// TIA Portal project "实验3_V20" (V20)

(* hardware
DEVICE "S7-300/ET200M station_1"  S7-300 station
   slot 0: "导轨_0"  Rail  6ES7 390-1***0-0AA0
   slot 2: "PLC_1"  CPU 314C-2 DP  6ES7 314-6CH04-0AB0  V3.3
      slot 0: "MPI 接口_1"  MPI
      slot 1: "DP 接口_1"  DP
      slot 2: "DI 24/DO 16_1"  DI24/DO16
      slot 3: "AI 5/AO 2_1"  AI5/AO2
      slot 4: "计数_1"  Counter
      slot 5: "定位_1"  Positioning
*)

// ===== PLC "PLC_1"  CPU 314C-2 DP =====

VAR_GLOBAL   // PLC tag table "默认变量表"
   "启动开关" AT %I0.0 : Bool;
   "光电传感器1" AT %I0.1 : Bool;
   "光电传感器2" AT %I0.2 : Bool;
   "光电传感器3" AT %I0.3 : Bool;
   "光电传感器4" AT %I0.4 : Bool;
   "电机正转" AT %Q4.1 : Bool;
   "电机反转" AT %Q4.2 : Bool;
   "位置1" AT %Q4.3 : Bool;
   "位置2" AT %Q4.4 : Bool;
   "位置3" AT %Q4.5 : Bool;
END_VAR

DATA_BLOCK "流程_DB"   // DB1
{ S7_Optimized_Access := 'FALSE' }
VERSION : 0.1
// stored: InstanceOfName 流程
"流程"
BEGIN
END_DATA_BLOCK

FUNCTION_BLOCK "流程"   // FB1, GRAPH
{ S7_Optimized_Access := 'FALSE' }
VERSION : 0.1
   VAR_INPUT
      OFF_SQ : Bool := false;   // 关闭顺控器
      INIT_SQ : Bool := false;   // 将顺序设置为初始状态
      ACK_EF : Bool := false;   // 确认所有的错误和故障
      S_PREV : Bool := false;   // 在S_NO输出参数中显示前导步
      S_NEXT : Bool := false;   // 在S_NO输出参数中显示后续步。
      SW_AUTO : Bool := false;   // 自动模式
      SW_TAP : Bool := false;   // 半自动/转换条件切换
      SW_TOP : Bool := false;   // 半自动/忽略转换条件
      SW_MAN : Bool := false;   // 手动模式
      S_SEL : Int := 0;   // 选择要在 S_NO中输出的步。
      S_ON : Bool := false;   // 激活S_NO 中显示的步。
      S_OFF : Bool := false;   // 禁用 S_NO 中标识的步
      T_PUSH : Bool := false;   // 允许在半自动模式下跳过转换条件。
   END_VAR
   VAR_OUTPUT
      S_NO : Int := 0;   // 步编号
      S_MORE : Bool := false;   // 更多步可用，并可在S_NO中显示。
      S_ACTIVE : Bool := false;   // 在S_NO 中显示的步是激活的。
      ERR_FLT : Bool := false;   // 互锁条件或监控条件组出错
      AUTO_ON : Bool := false;   // 当前为自动模式
      TAP_ON : Bool := false;   // 已启用SW_TAP模式。
      TOP_ON : Bool := false;   // 启用半自动模式/忽略转换条件。
      MAN_ON : Bool := false;   // 已启用手动模式。
   END_VAR
   VAR
      SWITCH : Array[0..0] of DWord;
      SW_SQTS : Array[0..7] of Byte;
      SW_ADDR : Word := 16#A;
      G7T_0 : GraphTransition;
      G7S_0 : GraphStep;
      PRE_CRIT : Array[0..0] of DWord;
      POST_CRIT : Array[0..0] of DWord;
      TVX : Array[0..2] of Byte;
      TTX : Array[0..2] of Byte;
      TSX : Array[0..2] of Byte;
      S00X : Array[0..2] of Byte;
      SOFFX : Array[0..2] of Byte;
      SONX : Array[0..2] of Byte;
      SAX : Array[0..2] of Byte;
      SERRX : Array[0..8] of Byte;
      SMX : Array[0..8] of Byte;
      S0X : Array[0..8] of Byte;
      S1X : Array[0..8] of Byte;
      S_DISPLAY : Int;   // 输出参数 S_NO 的内部显示
      S_SEL_OLD : Int;   // S_SEL 中的上一个值
      S_DISPIDX : Byte;   // S_NO 中步的索引
      T_DISPIDX : Byte;   // T_NO中转换条件的索引。
      MOPEDGE : Struct
         AUTO : Bool := false;
         MAN : Bool := false;
         TAP : Bool := false;
         TOP : Bool := false;
         ACK_S : Bool := false;
         REG_S : Bool := false;
         T_PREV : Bool := false;
         T_NEXT : Bool := false;
         LOCK : Bool := false;
         SUP : Bool := false;
         ACKREQ : Bool := false;
         SSKIP : Bool := false;
         OFF : Bool := false;
         INIT : Bool := false;
         HALT : Bool := false;
         TMS_HALT : Bool := false;
         OPS_ZERO : Bool := false;
         SACT_DISP : Bool := false;
         SEF_DISP : Bool := false;
         SALL_DISP : Bool := false;
         S_PREV : Bool := false;
         S_NEXT : Bool := false;
         S_SELOK : Bool := false;
         S_ON : Bool := false;
         S_OFF : Bool := false;
         T_PUSH : Bool := false;
         REG : Bool := false;
         ACK : Bool := false;
         IL_PERM : Bool := false;
         T_PERM : Bool := false;
         ILP_MAN : Bool := false;
      END_STRUCT;
      MOP : Struct   // 模式
         AUTO : Bool := true;   // 状态：自动模式
         MAN : Bool := false;   // 状态：手动模式
         TAP : Bool := false;   // 状态：半自动模式/手动切换
         TOP : Bool := false;   // 状态：半自动模式/忽略转换条件
         ACK_S : Bool := false;   // 请求：确认在参数S_NO 中显示的步。
         REG_S : Bool := false;   // 请求：记录 S_NO 中标识的步
         T_PREV : Bool := false;   // 请求：输出 T_NO 中上一个有效的转换条件
         T_NEXT : Bool := false;   // 请求：输出 T_NO 中下一个有效的转换条件
         LOCK : Bool := true;   // 状态：互锁已启用
         SUP : Bool := true;   // 状态：监控已启用
         ACKREQ : Bool := true;   // 状态：需要进行确认
         SSKIP : Bool := false;   // 状态：启用“忽略步”
         OFF : Bool := false;   // 请求：取消激活所有步
         INIT : Bool := true;   // 请求：将顺控器置位为初始状态
         HALT : Bool := false;   // 状态：顺控器已停止
         TMS_HALT : Bool := false;   // 状态：暂停所有内部定时器
         OPS_ZERO : Bool := false;   // 状态：将所有由 N、L 和 D 处理的操作数设置为 0
         SACT_DISP : Bool := true;   // 状态：仅显示活动步
         SEF_DISP : Bool := false;   // 状态：仅显示有错误的步和被中断的步。
         SALL_DISP : Bool := false;   // 状态：显示所有步
         S_PREV : Bool := false;   // 请求：在参数 S_NO 中输出前导步。
         S_NEXT : Bool := false;   // 请求：显示 S_NO 中的下一步 (NEXT_STEP)
         S_SELOK : Bool := false;   // 请求：从 SE_SEL 在 S_NO 处输出步编号
         S_ON : Bool := false;   // 请求：激活 S_NO 中标识的步
         S_OFF : Bool := false;   // 请求：取消激活 S_NO 中标识的步
         T_PUSH : Bool := false;   // 请求：启用转换条件进行切换
         REG : Bool := false;   // 请求：记录所有互锁条件和监控错误
         ACK : Bool := false;   // 请求：确认所有互锁条件和监控错误
         IL_PERM : Bool := false;   // 状态：总是处理所有互锁条件
         T_PERM : Bool := false;   // 状态： 总是处理所有转化条件
         ILP_MAN : Bool := false;   // 状态：手动模式下总是处理所有互锁条件
      END_STRUCT;
      TICKS : Struct   // 时钟速度
         DELTA : Time := T#0ms;   // 两个周期间的时间差
         OLD : Time := T#0ms;   // 上一次循环中的 10 ms 时钟计数值
         NEW : Time := T#0ms;   // 循环中时钟计数值为 10 ms
      END_STRUCT;
      SQ_FLAGS : Struct   // 顺序位存储器
         ERR_FLT : Bool := false;   // 互锁条件和监控条件组出错
         ERROR : Bool := false;   // 互锁条件组错误
         FAULT : Bool := false;   // 监视组错误
         RT_FAIL : Bool := false;   // 运行错误
         NO_SNO : Bool := false;   // 未找到所请求的步号
         NF_OFL : Bool := false;   // 溢出：ON 或 OFF 请求过多
         SA_OFL : Bool := false;   // 溢出：活动步过多。
         TV_OFL : Bool := false;   // 溢出：有效的转换条件过多
         MSG_OFL : Bool := false;   // 溢出：对于 ALARM_S 没有足够的系统资源
         NO_SWI : Bool := false;   // 在此循环中请勿切换
         CYC_OP : Bool := false;   // 初始化之后，循环顺序执行
         AS_MSG : Bool := true;   // 通过指令激活或取消激活运行期间报警。
         AS_SEND : Bool := false;   // 通过 WR_USMSG 发送报警或仅显示诊断缓冲区中。
         SQ_BUSY : Bool := false;   // 顺序处理的内部边沿位存储器。
         SA_BUSY : Bool := false;   // 顺序处理的内部边沿位存储器。
         AS_SIG : Bool := false;   // Alarm_S 和 Alarm_SQ 报警的边沿位存储器。
      END_STRUCT;
      S_PTR : DWord := 16#4C0;
      S_PTR2 : DWord := 16#0;
      S_PTR3 : DWord := 16#ED0;
      S_PTR4 : DWord := 16#E80;
      T_PTR : DWord := 16#E30;
      C_AR2 : DWord := 16#0;
      M_FBDB : DWord := 16#10000;
      M_SNO : Word := 16#0;
      M_EVID : Word := 16#0;
      M_EVIL : C_Alarm_s;
      M_EVSV : C_Alarm_s;
      M_EV : DWord := 16#D80;
      CRIT : Array[0..31] of Bool;
      S_START : Byte := 16#0;
      S_IDX : Byte := 16#0;
      S_INT : Int := 72;
      S_TMP : Byte := 16#0;
      T_START : Byte := 16#0;
      T_IDX : Byte := 16#0;
      T_TMP : Byte := 16#0;
      T_TMP2 : Byte := 16#00;
      TV_POT : Byte := 16#06;
      RETURN1 : Byte := 16#0;
      RETURN2 : Byte := 16#0;
      SINI : Array[0..2] of Byte;
      LSTT : Array[0..7] of Byte;
      ATAJ : Array[0..7] of Byte;
      ATAB : Array[0..7] of Byte;
      PSTT : Array[0..7] of Byte;
      NSTT : Array[0..7] of Byte;
      ASSJ : Array[0..7] of Byte;
      ASSB : Array[0..7] of Byte;
      PTTS : Array[0..7] of Byte;
      NTTS : Array[0..7] of Byte;
      PRE_CNT : Word := 16#1;
      POST_CNT : Word := 16#1;
      ADR_COND : Word := 16#0;
      MAX_TVAL : Byte := 16#1;
      MAX_SACT : Byte := 16#1;
      MAX_CRIT : Byte := 16#4;
      T_CNT : Byte := 16#7;
      SUP_CNT : Byte := 16#0;
      LOCK_CNT : Byte := 16#0;
      S_CNT : Byte := 16#7;
      SQ_CNT : Byte := 16#1;
      PRS_INPAR : DWord := 16#E000FEC8;
      PRS_OUTPAR : DWord := 16#E000800F;
      GC_FLAGS : Struct
         T_MACH : Byte := 16#EB;
         COND_ED : Byte := 16#E3;
         W_LEVEL : Byte := 16#D5;
         FB_IF : Byte := 16#FA;
         AS_MSG : Word := 16#404;
         SSB : Word := 16#108;
         DILG : Word := 16#2B0;
         ADDR_T0 : Word := 16#18;
         CRIT_AVAIL : Bool := false;
         SSKIP_AVAIL : Bool := true;
         SSKIP_ON : Bool := false;
         ACK_REQ : Bool := true;
         SYNC_AVAIL : Bool := true;
         ILP_MAN : Bool := false;
         SWM_LOCKED : Bool := false;
         SAVE_SW : Bool := true;
      END_STRUCT;
      G7_FBMARK : Byte := 16#3C;
      G7_RELEASE : Byte := 16#3C;
      G7_ID2 : Byte := 16#37;
      G7_ID1 : Byte := 16#47;
   END_VAR
   VAR_TEMP
      流程结束计时 : Bool;
   END_VAR
   // SW_SQTS[0] := 16#1;
   // TVX[0] := 16#1;
   // TTX[0] := 16#1;
   // TSX[0] := 16#1;
   // S00X[0] := 16#1;
   // SOFFX[0] := 16#1;
   // SONX[0] := 16#1;
   // SAX[0] := 16#1;
   // SERRX[0] := 16#1;
   // SMX[0] := 16#1;
   // S0X[0] := 16#1;
   // S1X[0] := 16#1;
   // SINI[0] := 16#2;
   // SINI[1] := 16#1;
   // SINI[2] := 0;
   // LSTT[0] := 0;
   // LSTT[1] := 0;
   // LSTT[2] := 0;
   // LSTT[3] := 0;
   // LSTT[4] := 0;
   // LSTT[5] := 0;
   // LSTT[6] := 0;
   // LSTT[7] := 16#1;
   // ATAJ[0] := 0;
   // ATAJ[1] := 16#1;
   // ATAJ[2] := 16#2;
   // ATAJ[3] := 16#3;
   // ATAJ[4] := 16#4;
   // ATAJ[5] := 16#5;
   // ATAJ[6] := 16#6;
   // ATAJ[7] := 16#7;
   // ATAB[0] := 0;
   // ATAB[1] := 16#1;
   // ATAB[2] := 16#2;
   // ATAB[3] := 16#3;
   // ATAB[4] := 16#4;
   // ATAB[5] := 16#5;
   // ATAB[6] := 16#6;
   // ATAB[7] := 16#7;
   // PSTT[0] := 0;
   // PSTT[1] := 16#1;
   // PSTT[2] := 16#2;
   // PSTT[3] := 16#3;
   // PSTT[4] := 16#4;
   // PSTT[5] := 16#5;
   // PSTT[6] := 16#6;
   // PSTT[7] := 16#7;
   // NSTT[0] := 16#1;
   // NSTT[1] := 16#2;
   // NSTT[2] := 16#3;
   // NSTT[3] := 16#4;
   // NSTT[4] := 16#5;
   // NSTT[5] := 16#6;
   // NSTT[6] := 16#7;
   // NSTT[7] := 16#1;
   // ASSJ[0] := 0;
   // ASSJ[1] := 16#1;
   // ASSJ[2] := 16#2;
   // ASSJ[3] := 16#3;
   // ASSJ[4] := 16#4;
   // ASSJ[5] := 16#5;
   // ASSJ[6] := 16#6;
   // ASSJ[7] := 16#7;
   // ASSB[0] := 0;
   // ASSB[1] := 16#1;
   // ASSB[2] := 16#2;
   // ASSB[3] := 16#3;
   // ASSB[4] := 16#4;
   // ASSB[5] := 16#5;
   // ASSB[6] := 16#6;
   // ASSB[7] := 16#7;
   // PTTS[0] := 0;
   // PTTS[2] := 16#1;
   // PTTS[3] := 16#2;
   // PTTS[4] := 16#3;
   // PTTS[5] := 16#4;
   // PTTS[6] := 16#5;
   // PTTS[7] := 16#6;
   // NTTS[0] := 0;
   // NTTS[1] := 16#1;
   // NTTS[2] := 16#2;
   // NTTS[3] := 16#3;
   // NTTS[4] := 16#4;
   // NTTS[5] := 16#5;
   // NTTS[6] := 16#6;
   // NTTS[7] := 16#7;
BEGIN
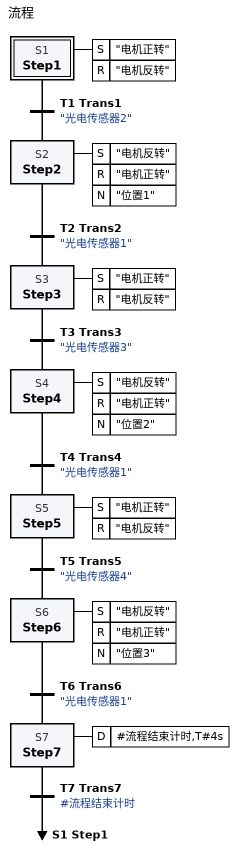
   // sequencer 1
   INITIAL_STEP Step1:   // S1
              S    "电机正转"
              R    "电机反转"
   END_STEP
   TRANSITION Trans1 FROM Step1 TO Step2   // T1
      := "光电传感器2";
   END_TRANSITION
   STEP Step2:   // S2
              S    "电机反转"
              R    "电机正转"
              N    "位置1"
   END_STEP
   TRANSITION Trans2 FROM Step2 TO Step3   // T2
      := "光电传感器1";
   END_TRANSITION
   STEP Step3:   // S3
              S    "电机正转"
              R    "电机反转"
   END_STEP
   TRANSITION Trans3 FROM Step3 TO Step4   // T3
      := "光电传感器3";
   END_TRANSITION
   STEP Step4:   // S4
              S    "电机反转"
              R    "电机正转"
              N    "位置2"
   END_STEP
   TRANSITION Trans4 FROM Step4 TO Step5   // T4
      := "光电传感器1";
   END_TRANSITION
   STEP Step5:   // S5
              S    "电机正转"
              R    "电机反转"
   END_STEP
   TRANSITION Trans5 FROM Step5 TO Step6   // T5
      := "光电传感器4";
   END_TRANSITION
   STEP Step6:   // S6
              S    "电机反转"
              R    "电机正转"
              N    "位置3"
   END_STEP
   TRANSITION Trans6 FROM Step6 TO Step7   // T6
      := "光电传感器1";
   END_TRANSITION
   STEP Step7:   // S7
              D    #流程结束计时,T#4s
   END_STEP
   TRANSITION Trans7 FROM Step7 TO Step1   // T7, jump
      := #流程结束计时;
   END_TRANSITION
END_FUNCTION_BLOCK

ORGANIZATION_BLOCK "Main"   // OB1, LAD
TITLE = "Main Program Sweep (Cycle)"
{ S7_Optimized_Access := 'FALSE' }
VERSION : 0.1
   VAR_TEMP
      OB1_EV_CLASS : Byte;   // Bits 0-3 = 1 (Coming event), Bits 4-7 = 1 (Event class 1)
      OB1_SCAN_1 : Byte;   // 1 (Cold restart scan 1 of OB 1), 3 (Scan 2-n of OB 1)
      OB1_PRIORITY : Byte;   // Priority of OB Execution
      OB1_OB_NUMBR : Byte;   // 1 (Organization block 1, OB1)
      OB1_RESERVED_1 : Byte;   // Reserved for system
      OB1_RESERVED_2 : Byte;   // Reserved for system
      OB1_PREV_CYCLE : Int;   // Cycle time of previous OB1 scan (milliseconds)
      OB1_MIN_CYCLE : Int;   // Minimum cycle time of OB1 (milliseconds)
      OB1_MAX_CYCLE : Int;   // Maximum cycle time of OB1 (milliseconds)
      OB1_DATE_TIME : Date_And_Time;   // Date and time OB1 started
   END_VAR
BEGIN

REGION Network 1
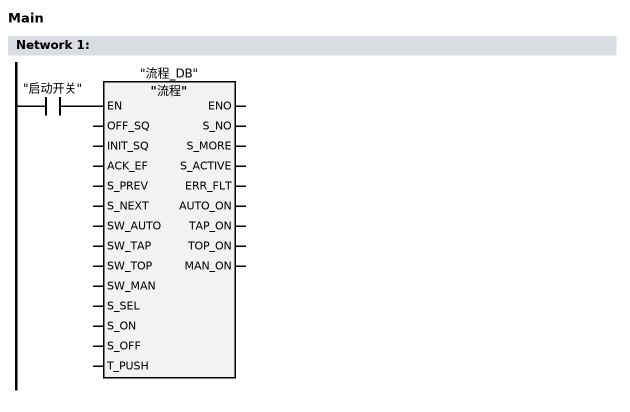
   RUNG wire#powerrail
      Contact( "启动开关" )
      "流程_DB"(OFF_SQ :=, INIT_SQ :=, ACK_EF :=, S_PREV :=, S_NEXT :=, SW_AUTO :=, SW_TAP :=, SW_TOP :=, SW_MAN :=, S_SEL :=, S_ON :=, S_OFF :=, T_PUSH :=, S_NO =>, S_MORE =>, S_ACTIVE =>, ERR_FLT =>, AUTO_ON =>, TAP_ON =>, TOP_ON =>, MAN_ON =>)
   END_RUNG
   // the same network as SCL:
   IF "启动开关" THEN
       "流程_DB"();   // "流程"
   END_IF;
END_REGION
END_ORGANIZATION_BLOCK